INTERFACE PUBLIC StartingCommands EXTENDS RunningStateCommands, ActionStateCommands, HoldableStateCommands

END_INTERFACE

(* stored: Version 1.1.0.1, ProductVersion 3.1.4026.18
   Itf StartingCommands: Id {dbee54f7-1ba1-0294-0b8c-497189d1fd31} *)
